// TIA Portal V18 program export: 1 tag tables, 0 data types, 0 data blocks, 1 code blocks (in call order from the OBs), 0 instance data blocks

VAR_GLOBAL   // PLC tag table "Default tag table"
   MOTOR_OUTPUT AT %M0.0 : Bool;
   MOTOR_START AT %M0.1 : Bool;
   MOTOR_STOP AT %M0.2 : Bool;
END_VAR

ORGANIZATION_BLOCK "Main"   // OB1, LAD, ProgramCycle
TITLE = "Main Program Sweep (Cycle)"
{ S7_Optimized_Access := 'TRUE' }
VERSION : 0.1
// stored: AutoNumber true, IsIECCheckEnabled false, SetENOAutomatically false
BEGIN

REGION Network 1 (SCL)
   "MOTOR_OUTPUT" := ("MOTOR_OUTPUT" OR "MOTOR_START") AND NOT "MOTOR_STOP";
END_REGION
END_ORGANIZATION_BLOCK
